INTERFACE ITF_0_BaseComponent

METHOD M_activate : BOOL
VAR_INPUT
END_VAR
END_METHOD

METHOD M_cleanup : BOOL
VAR_INPUT
END_VAR
END_METHOD

METHOD M_configure : BOOL
VAR_INPUT
END_VAR
END_METHOD

METHOD M_deactivate : BOOL
VAR_INPUT
END_VAR
END_METHOD

METHOD M_destroy : BOOL
VAR_INPUT
END_VAR
END_METHOD

METHOD M_shutdown : BOOL
VAR_INPUT
END_VAR
END_METHOD

METHOD onActivate : BOOL
VAR_INPUT
END_VAR
END_METHOD

METHOD onCleanup : BOOL
VAR_INPUT
END_VAR
END_METHOD

METHOD onConfigure : BOOL
VAR_INPUT
END_VAR
END_METHOD

METHOD onDeactivate : BOOL
VAR_INPUT
END_VAR
END_METHOD

METHOD onError : BOOL
VAR_INPUT
END_VAR
END_METHOD

METHOD onShutdown : BOOL
VAR_INPUT
END_VAR
END_METHOD

PROPERTY P_ID : UINT
GET
END_GET
SET
END_SET
END_PROPERTY

PROPERTY P_Name : String
GET
END_GET
END_PROPERTY

PROPERTY P_Path : String
GET
END_GET
END_PROPERTY

PROPERTY ABSTRACT P_State : eState
GET
END_GET
SET
END_SET
END_PROPERTY

END_INTERFACE

(* stored: Version 1.1.0.1, ProductVersion 3.1.4026.18
   Itf ITF_0_BaseComponent: Id {65885d39-4024-4344-a8ab-374a6ccc4c59}
   Folder Activities: Id {5e3aa71c-ec0e-47b3-8f33-f08f0fb99381}
   Folder Transitions: Id {6560e606-0171-480a-9918-20910c0e5bdf}
   Method M_activate: Id {421c2108-8179-4a12-ba41-35989c996212}
   Method M_cleanup: Id {2b58a7de-95d9-467c-85d1-db9dec921482}
   Method M_configure: Id {e50a6f49-0903-48ba-8271-1c9d1e1e510c}
   Method M_deactivate: Id {543d663f-3433-4738-bb10-46e710584fb3}
   Method M_destroy: Id {8dc262df-163a-4e11-9777-3fbb1a531627}
   Method M_shutdown: Id {d44b7757-327e-4329-96cc-8c180a9fb4f3}
   Method onActivate: Id {db5ccdf9-dda4-4656-8a40-44601294dbda}
   Method onCleanup: Id {aeb6ee92-c260-499d-8c85-ecf0511ec7d2}
   Method onConfigure: Id {5400f4d2-21c5-44f4-af11-064140524d3d}
   Method onDeactivate: Id {f1a21cdc-6225-4962-9570-04e28e96710c}
   Method onError: Id {6370aa46-a510-420e-b2b1-4a92b9216869}
   Method onShutdown: Id {6b29e55c-0bb5-4ed2-8d4c-29a2f4547848}
   Property P_ID: Id {fc62148d-d821-4a08-a5bf-6bdef92d59d5}
   Get Get: Id {c2985394-0d19-4b0e-a4c8-339d4db8e630}
   Set Set: Id {98424317-6db3-4da6-80d9-cb32dfe7d9a6}
   Property P_Name: Id {8e02e470-71da-44a6-a68f-092954d86151}
   Get Get: Id {7f1ff7dd-a478-4f29-885d-9677ae5d4a7e}
   Property P_Path: Id {755b1bdf-ea5e-45d8-b845-25d127de2ac2}
   Get Get: Id {bdac12b3-22bb-41f6-8039-bf0761521d8e}
   Property P_State: Id {4c5eddbd-3571-4017-85b4-cee88242beba}
   Get Get: Id {42aa47ea-f1d7-4040-ade8-b3efc7baaa84}
   Set Set: Id {1f4e04c9-7da1-43ff-a8c5-ecbad9f49fcd} *)
